Staubli VAL3: start.pgx

program start()
begin
  call Main(0)
end
